// Mitsubishi GX Works2 project: b3   PLC: Q03UDE

// global labels: Global1
VAR_GLOBAL
  startbut AT X40 : BOOL;
  stopbut AT X41 : BOOL;
  estop AT X42 : BOOL;
  qt AT Y50 : BOOL;
  qn AT Y51 : BOOL;
END_VAR

PROGRAM MAIN
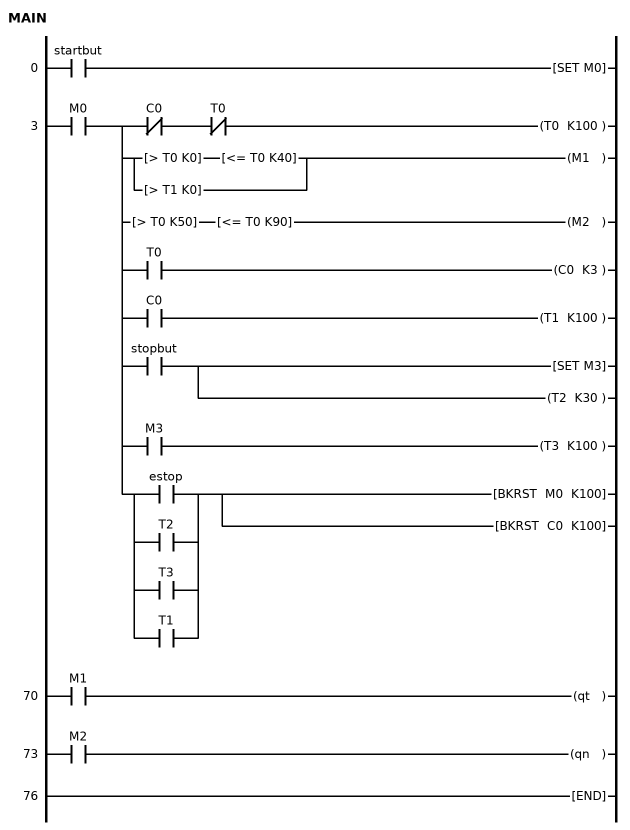
0     LD      startbut
      SET     M0
3     LD      M0
      MPS
      ANI     C0
      ANI     T0
      OUT     T0 K100
      MRD
      LD>     T0 K0
      AND<=   T0 K40
      OR>     T1 K0
      ANB
      OUT     M1
      MRD
      AND>    T0 K50
      AND<=   T0 K90
      OUT     M2
      MRD
      AND     T0
      OUT     C0 K3
      MRD
      AND     C0
      OUT     T1 K100
      MRD
      AND     stopbut
      SET     M3
      OUT     T2 K30
      MRD
      AND     M3
      OUT     T3 K100
      MPP
      LD      estop
      OR      T2
      OR      T3
      OR      T1
      ANB
      BKRST   M0 K100
      BKRST   C0 K100
70    LD      M1
      OUT     qt
73    LD      M2
      OUT     qn
76    END
END_PROGRAM
